// TIA Portal V17 export
// export: Created 2025-03-07T09:17:02.8526891Z, ExportSetting WithDefaults, DisplayName Totally Integrated Automation Portal, DisplayVersion V17 Update 8, DisplayName TIA Portal Openness, DisplayVersion V17 Update 8, DisplayName TIA Portal Version Control Interface, DisplayVersion V17, DisplayName SINAMICS Startdrive Advanced, DisplayVersion V17 SP2, DisplayName SINAMICS Startdrive G110M, G120, G120C, G120D, G120P, G115D, DisplayVersion V17 SP2, DisplayName SINAMICS Startdrive G130, G150, S120, S150, SINAMICS MV, S210, DisplayVersion V17 SP2, DisplayName STEP 7 Professional, DisplayVersion V17 Update 8, DisplayName SINUMERIK ONE STEP 7 Toolbox, DisplayVersion V17 Update 12, DisplayName SINUMERIK 840D sl STEP 7 Toolbox, DisplayVersion V17 Update 12, DisplayName STEP 7 Safety, DisplayVersion V17 Update 6, DisplayName WinCC Advanced, DisplayVersion V17 Update 8
FUNCTION "FC7454_QUALITY_FIRST_CYCLE_CLADDING" : Void   // FC7454, LAD
{ S7_Optimized_Access := 'FALSE' }
AUTHOR : ETXETAR
NAME : GM-QC
VERSION : 1.0
// stored: AutoNumber false, IsIECCheckEnabled false, SetENOAutomatically false, UDAEnableTagReadback false
   VAR_TEMP
      VALUE_0 : Real;
      AUX_FAULT : Bool;
   END_VAR
   VAR CONSTANT
      FC_NUMBER : DInt := 7454;
   END_VAR
   VAR_TEMP   // added for the SCL form of the ladder/FBD networks
      _w1 : Bool;
      _w2 : Bool;
   END_VAR
BEGIN

REGION Network 1: FIRST SCAN AUXILIARY SET
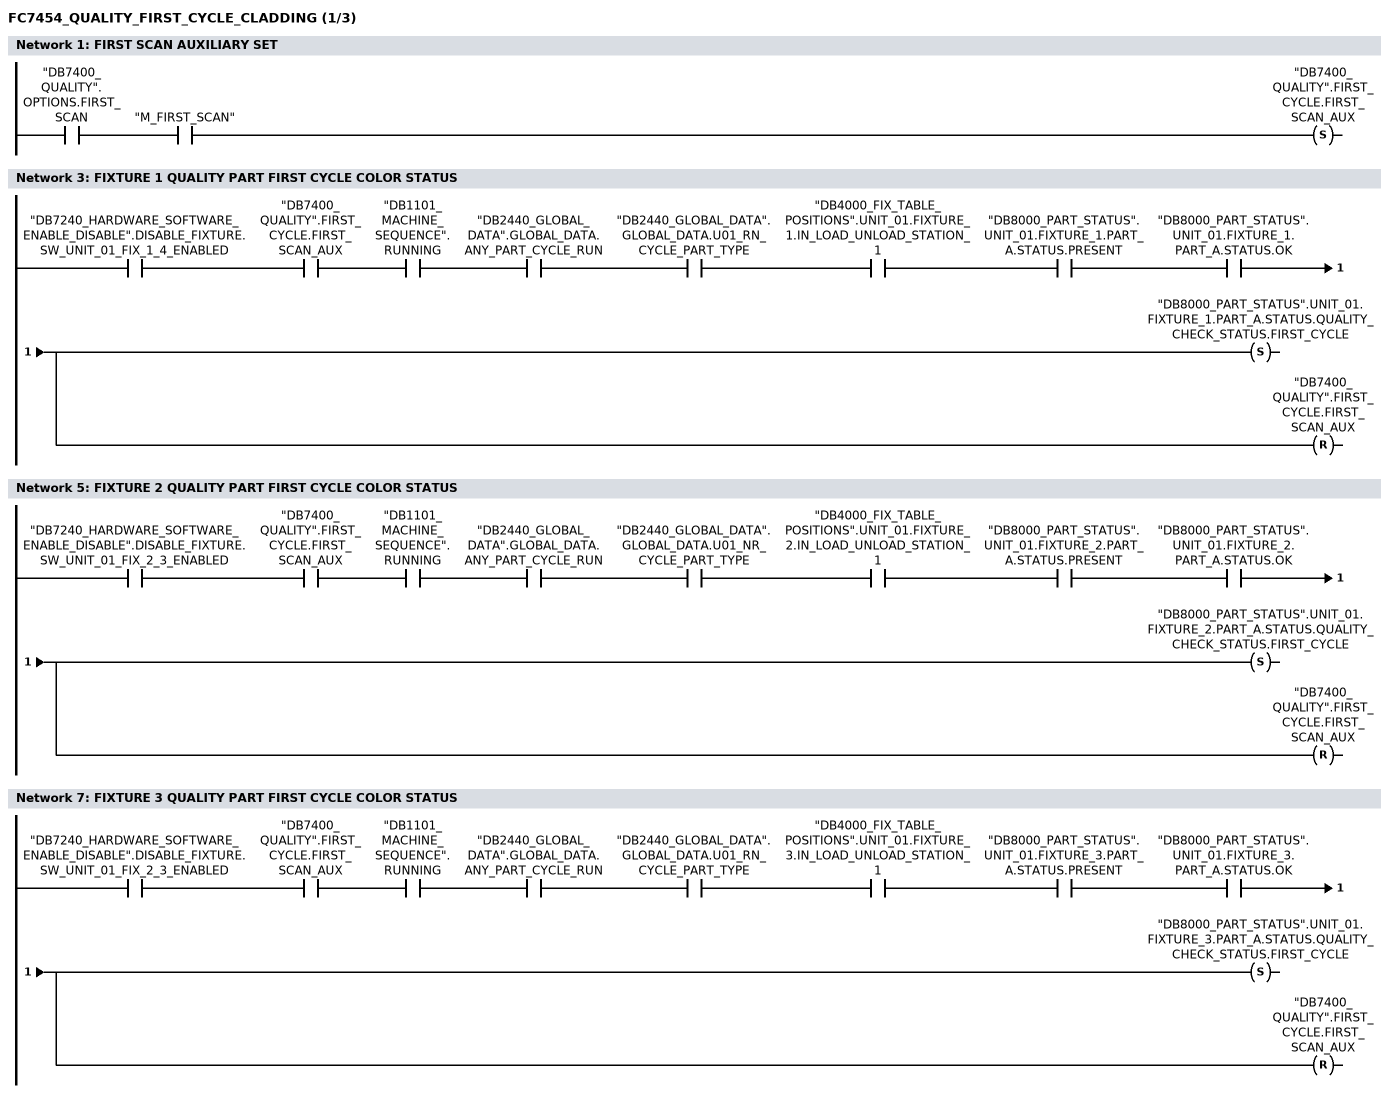
   RUNG wire#powerrail
      Contact( "DB7400_QUALITY".OPTIONS.FIRST_SCAN )
      Contact( "M_FIRST_SCAN" )
      S_Coil( "DB7400_QUALITY".FIRST_CYCLE.FIRST_SCAN_AUX )
   END_RUNG
   // the same network as SCL:
   IF "DB7400_QUALITY".OPTIONS.FIRST_SCAN AND "M_FIRST_SCAN" THEN
       "DB7400_QUALITY".FIRST_CYCLE.FIRST_SCAN_AUX := TRUE;
   END_IF;
END_REGION

REGION Network 2: /////_FIXTURE_1_/////
END_REGION

REGION Network 3: FIXTURE 1 QUALITY PART FIRST CYCLE COLOR STATUS
   RUNG wire#powerrail
      Contact( "DB7240_HARDWARE_SOFTWARE_ENABLE_DISABLE".DISABLE_FIXTURE.SW_UNIT_01_FIX_1_4_ENABLED )
      Contact( "DB7400_QUALITY".FIRST_CYCLE.FIRST_SCAN_AUX )
      Contact( "DB1101_MACHINE_SEQUENCE".RUNNING )
      Contact( "DB2440_GLOBAL_DATA".GLOBAL_DATA.ANY_PART_CYCLE_RUN )
      Contact( "DB2440_GLOBAL_DATA".GLOBAL_DATA.U01_RN_CYCLE_PART_TYPE )
      Contact( "DB4000_FIX_TABLE_POSITIONS".UNIT_01.FIXTURE_1.IN_LOAD_UNLOAD_STATION_1 )
      Contact( "DB8000_PART_STATUS".UNIT_01.FIXTURE_1.PART_A.STATUS.PRESENT )
      Contact( "DB8000_PART_STATUS".UNIT_01.FIXTURE_1.PART_A.STATUS.OK )
      wire#w1
      S_Coil( "DB8000_PART_STATUS".UNIT_01.FIXTURE_1.PART_A.STATUS.QUALITY_CHECK_STATUS.FIRST_CYCLE )
   END_RUNG
   RUNG wire#w1
      R_Coil( "DB7400_QUALITY".FIRST_CYCLE.FIRST_SCAN_AUX )
   END_RUNG
   // the same network as SCL:
   IF "DB7240_HARDWARE_SOFTWARE_ENABLE_DISABLE".DISABLE_FIXTURE.SW_UNIT_01_FIX_1_4_ENABLED AND "DB7400_QUALITY".FIRST_CYCLE.FIRST_SCAN_AUX AND "DB1101_MACHINE_SEQUENCE".RUNNING AND "DB2440_GLOBAL_DATA".GLOBAL_DATA.ANY_PART_CYCLE_RUN AND "DB2440_GLOBAL_DATA".GLOBAL_DATA.U01_RN_CYCLE_PART_TYPE AND "DB4000_FIX_TABLE_POSITIONS".UNIT_01.FIXTURE_1.IN_LOAD_UNLOAD_STATION_1 AND "DB8000_PART_STATUS".UNIT_01.FIXTURE_1.PART_A.STATUS.PRESENT AND "DB8000_PART_STATUS".UNIT_01.FIXTURE_1.PART_A.STATUS.OK THEN
       "DB8000_PART_STATUS".UNIT_01.FIXTURE_1.PART_A.STATUS.QUALITY_CHECK_STATUS.FIRST_CYCLE := TRUE;
       "DB7400_QUALITY".FIRST_CYCLE.FIRST_SCAN_AUX := FALSE;
   END_IF;
END_REGION

REGION Network 4: /////_FIXTURE_2_/////
END_REGION

REGION Network 5: FIXTURE 2 QUALITY PART FIRST CYCLE COLOR STATUS
   RUNG wire#powerrail
      Contact( "DB7240_HARDWARE_SOFTWARE_ENABLE_DISABLE".DISABLE_FIXTURE.SW_UNIT_01_FIX_2_3_ENABLED )
      Contact( "DB7400_QUALITY".FIRST_CYCLE.FIRST_SCAN_AUX )
      Contact( "DB1101_MACHINE_SEQUENCE".RUNNING )
      Contact( "DB2440_GLOBAL_DATA".GLOBAL_DATA.ANY_PART_CYCLE_RUN )
      Contact( "DB2440_GLOBAL_DATA".GLOBAL_DATA.U01_NR_CYCLE_PART_TYPE )
      Contact( "DB4000_FIX_TABLE_POSITIONS".UNIT_01.FIXTURE_2.IN_LOAD_UNLOAD_STATION_1 )
      Contact( "DB8000_PART_STATUS".UNIT_01.FIXTURE_2.PART_A.STATUS.PRESENT )
      Contact( "DB8000_PART_STATUS".UNIT_01.FIXTURE_2.PART_A.STATUS.OK )
      wire#w1
      S_Coil( "DB8000_PART_STATUS".UNIT_01.FIXTURE_2.PART_A.STATUS.QUALITY_CHECK_STATUS.FIRST_CYCLE )
   END_RUNG
   RUNG wire#w1
      R_Coil( "DB7400_QUALITY".FIRST_CYCLE.FIRST_SCAN_AUX )
   END_RUNG
   // the same network as SCL:
   IF "DB7240_HARDWARE_SOFTWARE_ENABLE_DISABLE".DISABLE_FIXTURE.SW_UNIT_01_FIX_2_3_ENABLED AND "DB7400_QUALITY".FIRST_CYCLE.FIRST_SCAN_AUX AND "DB1101_MACHINE_SEQUENCE".RUNNING AND "DB2440_GLOBAL_DATA".GLOBAL_DATA.ANY_PART_CYCLE_RUN AND "DB2440_GLOBAL_DATA".GLOBAL_DATA.U01_NR_CYCLE_PART_TYPE AND "DB4000_FIX_TABLE_POSITIONS".UNIT_01.FIXTURE_2.IN_LOAD_UNLOAD_STATION_1 AND "DB8000_PART_STATUS".UNIT_01.FIXTURE_2.PART_A.STATUS.PRESENT AND "DB8000_PART_STATUS".UNIT_01.FIXTURE_2.PART_A.STATUS.OK THEN
       "DB8000_PART_STATUS".UNIT_01.FIXTURE_2.PART_A.STATUS.QUALITY_CHECK_STATUS.FIRST_CYCLE := TRUE;
       "DB7400_QUALITY".FIRST_CYCLE.FIRST_SCAN_AUX := FALSE;
   END_IF;
END_REGION

REGION Network 6: /////_FIXTURE_3_/////
END_REGION

REGION Network 7: FIXTURE 3 QUALITY PART FIRST CYCLE COLOR STATUS
   RUNG wire#powerrail
      Contact( "DB7240_HARDWARE_SOFTWARE_ENABLE_DISABLE".DISABLE_FIXTURE.SW_UNIT_01_FIX_2_3_ENABLED )
      Contact( "DB7400_QUALITY".FIRST_CYCLE.FIRST_SCAN_AUX )
      Contact( "DB1101_MACHINE_SEQUENCE".RUNNING )
      Contact( "DB2440_GLOBAL_DATA".GLOBAL_DATA.ANY_PART_CYCLE_RUN )
      Contact( "DB2440_GLOBAL_DATA".GLOBAL_DATA.U01_RN_CYCLE_PART_TYPE )
      Contact( "DB4000_FIX_TABLE_POSITIONS".UNIT_01.FIXTURE_3.IN_LOAD_UNLOAD_STATION_1 )
      Contact( "DB8000_PART_STATUS".UNIT_01.FIXTURE_3.PART_A.STATUS.PRESENT )
      Contact( "DB8000_PART_STATUS".UNIT_01.FIXTURE_3.PART_A.STATUS.OK )
      wire#w1
      S_Coil( "DB8000_PART_STATUS".UNIT_01.FIXTURE_3.PART_A.STATUS.QUALITY_CHECK_STATUS.FIRST_CYCLE )
   END_RUNG
   RUNG wire#w1
      R_Coil( "DB7400_QUALITY".FIRST_CYCLE.FIRST_SCAN_AUX )
   END_RUNG
   // the same network as SCL:
   IF "DB7240_HARDWARE_SOFTWARE_ENABLE_DISABLE".DISABLE_FIXTURE.SW_UNIT_01_FIX_2_3_ENABLED AND "DB7400_QUALITY".FIRST_CYCLE.FIRST_SCAN_AUX AND "DB1101_MACHINE_SEQUENCE".RUNNING AND "DB2440_GLOBAL_DATA".GLOBAL_DATA.ANY_PART_CYCLE_RUN AND "DB2440_GLOBAL_DATA".GLOBAL_DATA.U01_RN_CYCLE_PART_TYPE AND "DB4000_FIX_TABLE_POSITIONS".UNIT_01.FIXTURE_3.IN_LOAD_UNLOAD_STATION_1 AND "DB8000_PART_STATUS".UNIT_01.FIXTURE_3.PART_A.STATUS.PRESENT AND "DB8000_PART_STATUS".UNIT_01.FIXTURE_3.PART_A.STATUS.OK THEN
       "DB8000_PART_STATUS".UNIT_01.FIXTURE_3.PART_A.STATUS.QUALITY_CHECK_STATUS.FIRST_CYCLE := TRUE;
       "DB7400_QUALITY".FIRST_CYCLE.FIRST_SCAN_AUX := FALSE;
   END_IF;
END_REGION

REGION Network 8: /////_FIXTURE_4_/////
END_REGION

REGION Network 9: FIXTURE 4 QUALITY PART FIRST CYCLE COLOR STATUS
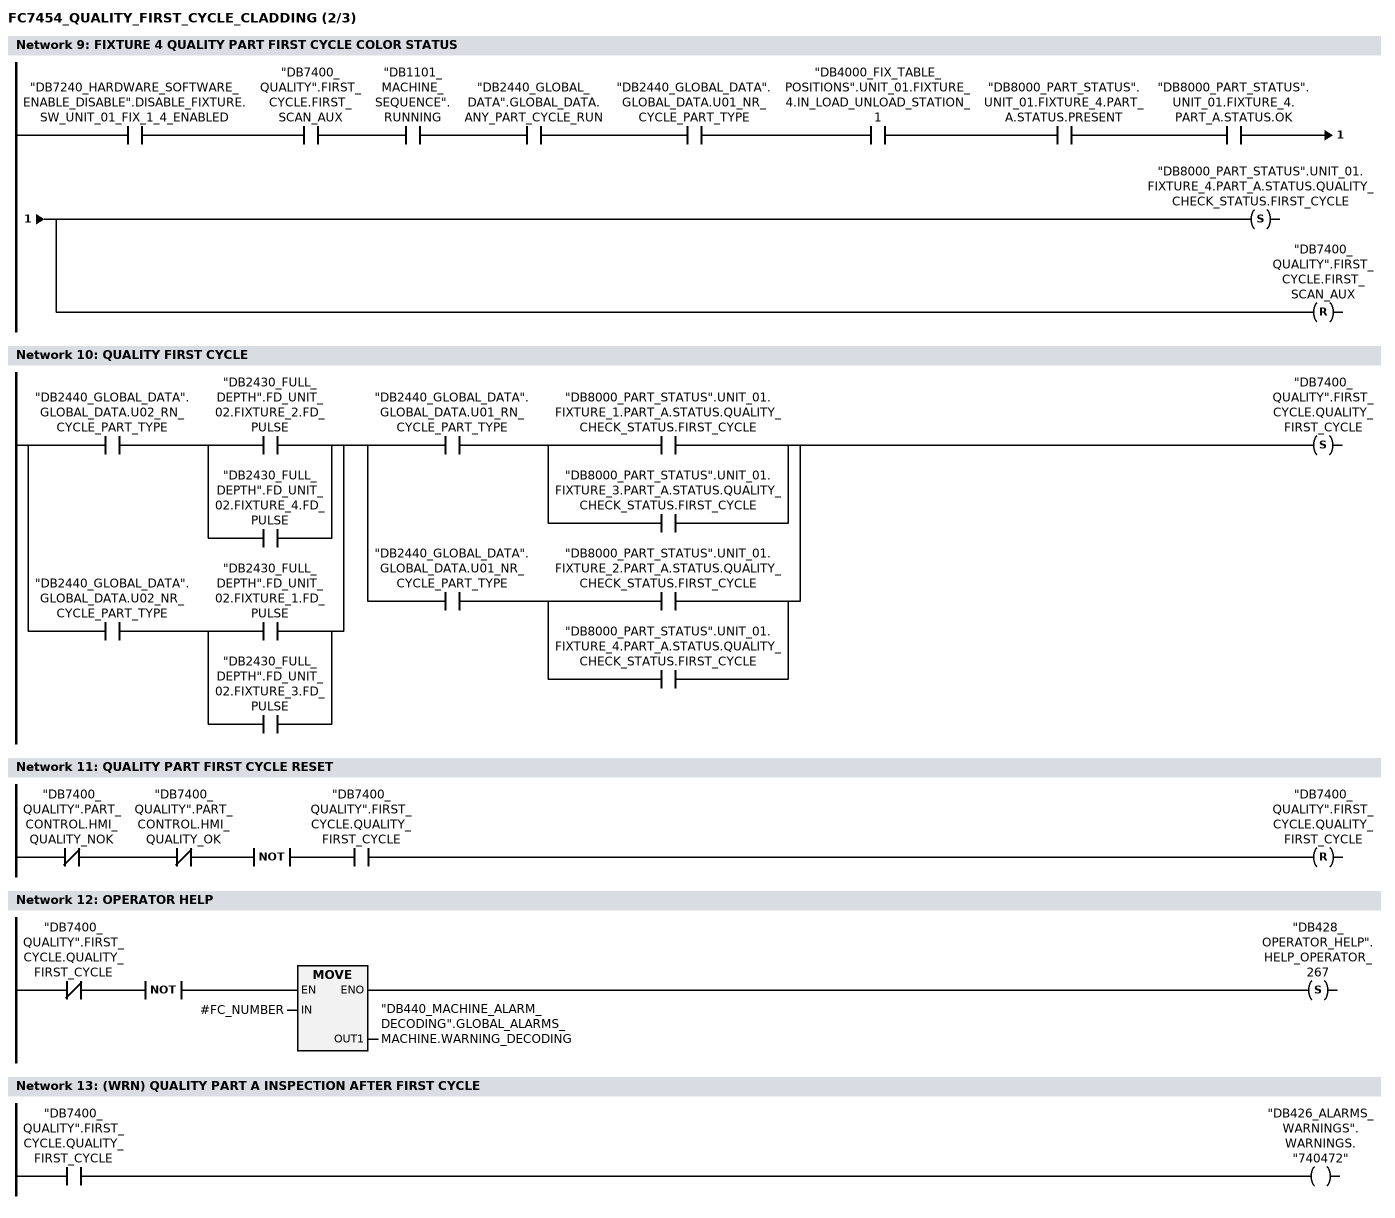
   RUNG wire#powerrail
      Contact( "DB7240_HARDWARE_SOFTWARE_ENABLE_DISABLE".DISABLE_FIXTURE.SW_UNIT_01_FIX_1_4_ENABLED )
      Contact( "DB7400_QUALITY".FIRST_CYCLE.FIRST_SCAN_AUX )
      Contact( "DB1101_MACHINE_SEQUENCE".RUNNING )
      Contact( "DB2440_GLOBAL_DATA".GLOBAL_DATA.ANY_PART_CYCLE_RUN )
      Contact( "DB2440_GLOBAL_DATA".GLOBAL_DATA.U01_NR_CYCLE_PART_TYPE )
      Contact( "DB4000_FIX_TABLE_POSITIONS".UNIT_01.FIXTURE_4.IN_LOAD_UNLOAD_STATION_1 )
      Contact( "DB8000_PART_STATUS".UNIT_01.FIXTURE_4.PART_A.STATUS.PRESENT )
      Contact( "DB8000_PART_STATUS".UNIT_01.FIXTURE_4.PART_A.STATUS.OK )
      wire#w1
      S_Coil( "DB8000_PART_STATUS".UNIT_01.FIXTURE_4.PART_A.STATUS.QUALITY_CHECK_STATUS.FIRST_CYCLE )
   END_RUNG
   RUNG wire#w1
      R_Coil( "DB7400_QUALITY".FIRST_CYCLE.FIRST_SCAN_AUX )
   END_RUNG
   // the same network as SCL:
   IF "DB7240_HARDWARE_SOFTWARE_ENABLE_DISABLE".DISABLE_FIXTURE.SW_UNIT_01_FIX_1_4_ENABLED AND "DB7400_QUALITY".FIRST_CYCLE.FIRST_SCAN_AUX AND "DB1101_MACHINE_SEQUENCE".RUNNING AND "DB2440_GLOBAL_DATA".GLOBAL_DATA.ANY_PART_CYCLE_RUN AND "DB2440_GLOBAL_DATA".GLOBAL_DATA.U01_NR_CYCLE_PART_TYPE AND "DB4000_FIX_TABLE_POSITIONS".UNIT_01.FIXTURE_4.IN_LOAD_UNLOAD_STATION_1 AND "DB8000_PART_STATUS".UNIT_01.FIXTURE_4.PART_A.STATUS.PRESENT AND "DB8000_PART_STATUS".UNIT_01.FIXTURE_4.PART_A.STATUS.OK THEN
       "DB8000_PART_STATUS".UNIT_01.FIXTURE_4.PART_A.STATUS.QUALITY_CHECK_STATUS.FIRST_CYCLE := TRUE;
       "DB7400_QUALITY".FIRST_CYCLE.FIRST_SCAN_AUX := FALSE;
   END_IF;
END_REGION

REGION Network 10: QUALITY FIRST CYCLE
   RUNG wire#powerrail
      Contact( "DB2440_GLOBAL_DATA".GLOBAL_DATA.U02_RN_CYCLE_PART_TYPE )
      wire#w1
      Contact( "DB2430_FULL_DEPTH".FD_UNIT_02.FIXTURE_2.FD_PULSE )
      wire#w2
      Contact( "DB2440_GLOBAL_DATA".GLOBAL_DATA.U01_RN_CYCLE_PART_TYPE )
      wire#w4
      Contact( "DB8000_PART_STATUS".UNIT_01.FIXTURE_1.PART_A.STATUS.QUALITY_CHECK_STATUS.FIRST_CYCLE )
      wire#w5
      S_Coil( "DB7400_QUALITY".FIRST_CYCLE.QUALITY_FIRST_CYCLE )
   END_RUNG
   RUNG wire#w1
      Contact( "DB2430_FULL_DEPTH".FD_UNIT_02.FIXTURE_4.FD_PULSE )
   END_RUNG wire#w2
   RUNG wire#powerrail
      Contact( "DB2440_GLOBAL_DATA".GLOBAL_DATA.U02_NR_CYCLE_PART_TYPE )
      wire#w3
      Contact( "DB2430_FULL_DEPTH".FD_UNIT_02.FIXTURE_1.FD_PULSE )
   END_RUNG wire#w2
   RUNG wire#w3
      Contact( "DB2430_FULL_DEPTH".FD_UNIT_02.FIXTURE_3.FD_PULSE )
   END_RUNG wire#w2
   RUNG wire#w4
      Contact( "DB8000_PART_STATUS".UNIT_01.FIXTURE_3.PART_A.STATUS.QUALITY_CHECK_STATUS.FIRST_CYCLE )
   END_RUNG wire#w5
   RUNG wire#w2
      Contact( "DB2440_GLOBAL_DATA".GLOBAL_DATA.U01_NR_CYCLE_PART_TYPE )
      wire#w6
      Contact( "DB8000_PART_STATUS".UNIT_01.FIXTURE_2.PART_A.STATUS.QUALITY_CHECK_STATUS.FIRST_CYCLE )
   END_RUNG wire#w5
   RUNG wire#w6
      Contact( "DB8000_PART_STATUS".UNIT_01.FIXTURE_4.PART_A.STATUS.QUALITY_CHECK_STATUS.FIRST_CYCLE )
   END_RUNG wire#w5
   // the same network as SCL:
   IF (("DB2440_GLOBAL_DATA".GLOBAL_DATA.U02_RN_CYCLE_PART_TYPE AND ("DB2430_FULL_DEPTH".FD_UNIT_02.FIXTURE_2.FD_PULSE OR "DB2430_FULL_DEPTH".FD_UNIT_02.FIXTURE_4.FD_PULSE)) OR ("DB2440_GLOBAL_DATA".GLOBAL_DATA.U02_NR_CYCLE_PART_TYPE AND ("DB2430_FULL_DEPTH".FD_UNIT_02.FIXTURE_1.FD_PULSE OR "DB2430_FULL_DEPTH".FD_UNIT_02.FIXTURE_3.FD_PULSE))) AND (("DB2440_GLOBAL_DATA".GLOBAL_DATA.U01_RN_CYCLE_PART_TYPE AND ("DB8000_PART_STATUS".UNIT_01.FIXTURE_1.PART_A.STATUS.QUALITY_CHECK_STATUS.FIRST_CYCLE OR "DB8000_PART_STATUS".UNIT_01.FIXTURE_3.PART_A.STATUS.QUALITY_CHECK_STATUS.FIRST_CYCLE)) OR ("DB2440_GLOBAL_DATA".GLOBAL_DATA.U01_NR_CYCLE_PART_TYPE AND ("DB8000_PART_STATUS".UNIT_01.FIXTURE_2.PART_A.STATUS.QUALITY_CHECK_STATUS.FIRST_CYCLE OR "DB8000_PART_STATUS".UNIT_01.FIXTURE_4.PART_A.STATUS.QUALITY_CHECK_STATUS.FIRST_CYCLE))) THEN
       "DB7400_QUALITY".FIRST_CYCLE.QUALITY_FIRST_CYCLE := TRUE;
   END_IF;
END_REGION

REGION Network 11: QUALITY PART FIRST CYCLE RESET
   RUNG wire#powerrail
      I_Contact( "DB7400_QUALITY".PART_CONTROL.HMI_QUALITY_NOK )
      I_Contact( "DB7400_QUALITY".PART_CONTROL.HMI_QUALITY_OK )
      Not()
      Contact( "DB7400_QUALITY".FIRST_CYCLE.QUALITY_FIRST_CYCLE )
      R_Coil( "DB7400_QUALITY".FIRST_CYCLE.QUALITY_FIRST_CYCLE )
   END_RUNG
   // the same network as SCL:
   IF NOT (NOT "DB7400_QUALITY".PART_CONTROL.HMI_QUALITY_NOK AND NOT "DB7400_QUALITY".PART_CONTROL.HMI_QUALITY_OK) AND "DB7400_QUALITY".FIRST_CYCLE.QUALITY_FIRST_CYCLE THEN
       "DB7400_QUALITY".FIRST_CYCLE.QUALITY_FIRST_CYCLE := FALSE;
   END_IF;
END_REGION

REGION Network 12: OPERATOR HELP
   RUNG wire#powerrail
      I_Contact( "DB7400_QUALITY".FIRST_CYCLE.QUALITY_FIRST_CYCLE )
      Not()
      { S7_GenerateENO := "TRUE" } Move(in := #FC_NUMBER, out1 => "DB440_MACHINE_ALARM_DECODING".GLOBAL_ALARMS_MACHINE.WARNING_DECODING)
      S_Coil( "DB428_OPERATOR_HELP".HELP_OPERATOR_267 )
   END_RUNG
   // the same network as SCL:
   // ENO of a box is taken as its EN; it also drops when the box reports an error
   IF NOT (NOT "DB7400_QUALITY".FIRST_CYCLE.QUALITY_FIRST_CYCLE) THEN
       "DB440_MACHINE_ALARM_DECODING".GLOBAL_ALARMS_MACHINE.WARNING_DECODING := #FC_NUMBER;
       "DB428_OPERATOR_HELP".HELP_OPERATOR_267 := TRUE;
   END_IF;
END_REGION

REGION Network 13: (WRN) QUALITY PART A INSPECTION AFTER FIRST CYCLE
   RUNG wire#powerrail
      Contact( "DB7400_QUALITY".FIRST_CYCLE.QUALITY_FIRST_CYCLE )
      Coil( "DB426_ALARMS_WARNINGS".WARNINGS."740472" )
   END_RUNG
   // the same network as SCL:
   "DB426_ALARMS_WARNINGS".WARNINGS."740472" := "DB7400_QUALITY".FIRST_CYCLE.QUALITY_FIRST_CYCLE;
END_REGION

REGION Network 14: QUALITY PART A FIRST CYCLE NOK ALARM
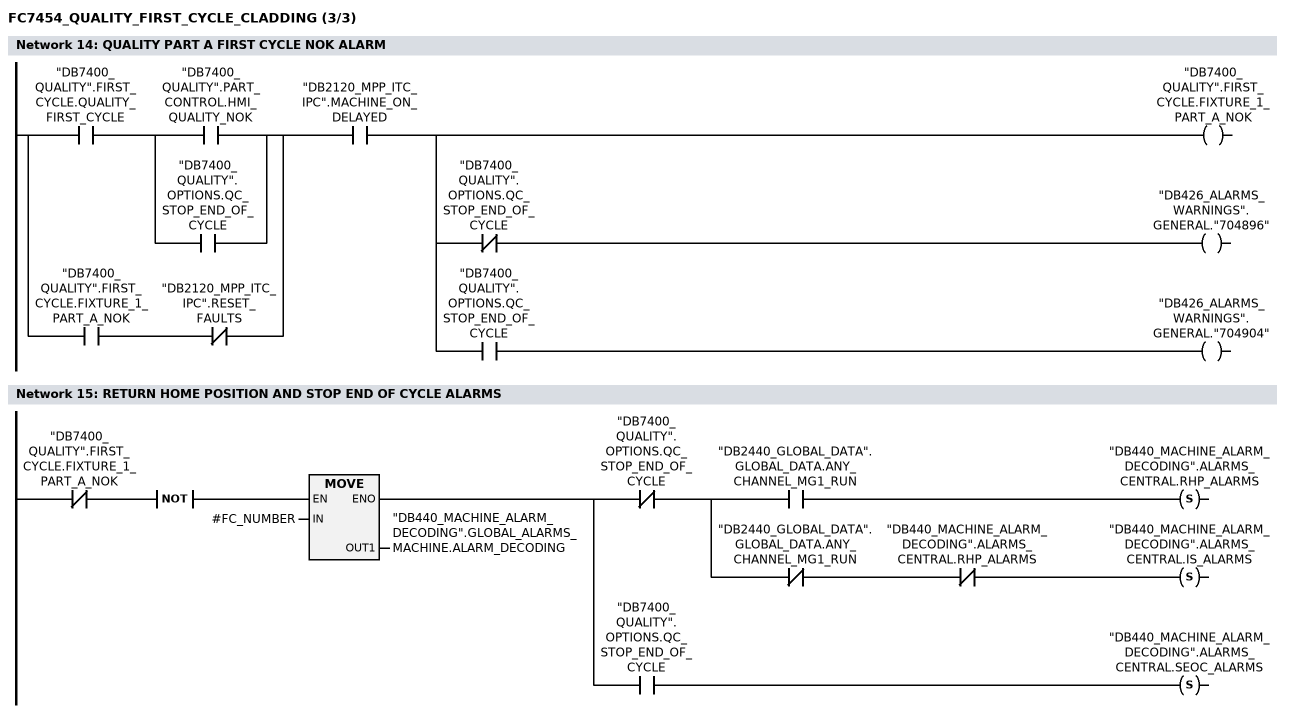
   RUNG wire#powerrail
      Contact( "DB7400_QUALITY".FIRST_CYCLE.QUALITY_FIRST_CYCLE )
      wire#w1
      Contact( "DB7400_QUALITY".PART_CONTROL.HMI_QUALITY_NOK )
      wire#w2
      Contact( "DB2120_MPP_ITC_IPC".MACHINE_ON_DELAYED )
      wire#w3
      Coil( "DB7400_QUALITY".FIRST_CYCLE.FIXTURE_1_PART_A_NOK )
   END_RUNG
   RUNG wire#w1
      Contact( "DB7400_QUALITY".OPTIONS.QC_STOP_END_OF_CYCLE )
   END_RUNG wire#w2
   RUNG wire#powerrail
      Contact( "DB7400_QUALITY".FIRST_CYCLE.FIXTURE_1_PART_A_NOK )
      I_Contact( "DB2120_MPP_ITC_IPC".RESET_FAULTS )
   END_RUNG wire#w2
   RUNG wire#w3
      I_Contact( "DB7400_QUALITY".OPTIONS.QC_STOP_END_OF_CYCLE )
      Coil( "DB426_ALARMS_WARNINGS".GENERAL."704896" )
   END_RUNG
   RUNG wire#w3
      Contact( "DB7400_QUALITY".OPTIONS.QC_STOP_END_OF_CYCLE )
      Coil( "DB426_ALARMS_WARNINGS".GENERAL."704904" )
   END_RUNG
   // the same network as SCL:
   "DB7400_QUALITY".FIRST_CYCLE.FIXTURE_1_PART_A_NOK := (("DB7400_QUALITY".FIRST_CYCLE.QUALITY_FIRST_CYCLE AND ("DB7400_QUALITY".PART_CONTROL.HMI_QUALITY_NOK OR "DB7400_QUALITY".OPTIONS.QC_STOP_END_OF_CYCLE)) OR ("DB7400_QUALITY".FIRST_CYCLE.FIXTURE_1_PART_A_NOK AND NOT "DB2120_MPP_ITC_IPC".RESET_FAULTS)) AND "DB2120_MPP_ITC_IPC".MACHINE_ON_DELAYED;
   "DB426_ALARMS_WARNINGS".GENERAL."704896" := "DB7400_QUALITY".FIRST_CYCLE.FIXTURE_1_PART_A_NOK AND NOT "DB7400_QUALITY".OPTIONS.QC_STOP_END_OF_CYCLE;
   "DB426_ALARMS_WARNINGS".GENERAL."704904" := "DB7400_QUALITY".FIRST_CYCLE.FIXTURE_1_PART_A_NOK AND "DB7400_QUALITY".OPTIONS.QC_STOP_END_OF_CYCLE;
END_REGION

REGION Network 15: RETURN HOME POSITION AND STOP END OF CYCLE ALARMS
   RUNG wire#powerrail
      I_Contact( "DB7400_QUALITY".FIRST_CYCLE.FIXTURE_1_PART_A_NOK )
      Not()
      { S7_GenerateENO := "TRUE" } Move(in := #FC_NUMBER, out1 => "DB440_MACHINE_ALARM_DECODING".GLOBAL_ALARMS_MACHINE.ALARM_DECODING)
      wire#w1
      I_Contact( "DB7400_QUALITY".OPTIONS.QC_STOP_END_OF_CYCLE )
      wire#w2
      Contact( "DB2440_GLOBAL_DATA".GLOBAL_DATA.ANY_CHANNEL_MG1_RUN )
      S_Coil( "DB440_MACHINE_ALARM_DECODING".ALARMS_CENTRAL.RHP_ALARMS )
   END_RUNG
   RUNG wire#w2
      I_Contact( "DB2440_GLOBAL_DATA".GLOBAL_DATA.ANY_CHANNEL_MG1_RUN )
      I_Contact( "DB440_MACHINE_ALARM_DECODING".ALARMS_CENTRAL.RHP_ALARMS )
      S_Coil( "DB440_MACHINE_ALARM_DECODING".ALARMS_CENTRAL.IS_ALARMS )
   END_RUNG
   RUNG wire#w1
      Contact( "DB7400_QUALITY".OPTIONS.QC_STOP_END_OF_CYCLE )
      S_Coil( "DB440_MACHINE_ALARM_DECODING".ALARMS_CENTRAL.SEOC_ALARMS )
   END_RUNG
   // the same network as SCL:
   // ENO of a box is taken as its EN; it also drops when the box reports an error
   #_w1 := NOT (NOT "DB7400_QUALITY".FIRST_CYCLE.FIXTURE_1_PART_A_NOK);
   IF #_w1 THEN "DB440_MACHINE_ALARM_DECODING".GLOBAL_ALARMS_MACHINE.ALARM_DECODING := #FC_NUMBER; END_IF;
   #_w2 := #_w1 AND NOT "DB7400_QUALITY".OPTIONS.QC_STOP_END_OF_CYCLE;
   IF #_w2 AND "DB2440_GLOBAL_DATA".GLOBAL_DATA.ANY_CHANNEL_MG1_RUN THEN
       "DB440_MACHINE_ALARM_DECODING".ALARMS_CENTRAL.RHP_ALARMS := TRUE;
   END_IF;
   IF #_w2 AND NOT "DB2440_GLOBAL_DATA".GLOBAL_DATA.ANY_CHANNEL_MG1_RUN AND NOT "DB440_MACHINE_ALARM_DECODING".ALARMS_CENTRAL.RHP_ALARMS THEN
       "DB440_MACHINE_ALARM_DECODING".ALARMS_CENTRAL.IS_ALARMS := TRUE;
   END_IF;
   IF #_w1 AND "DB7400_QUALITY".OPTIONS.QC_STOP_END_OF_CYCLE THEN
       "DB440_MACHINE_ALARM_DECODING".ALARMS_CENTRAL.SEOC_ALARMS := TRUE;
   END_IF;
END_REGION
END_FUNCTION
